FUNCTION_BLOCK POU IMPLEMENTS ITcTask
VAR_INPUT
END_VAR
VAR_OUTPUT
END_VAR
VAR
END_VAR

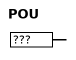
// ???: input not connected

{attribute 'TcTypeSystem'}
{attribute 'no-analysis'}
{attribute 'c++_compatible'}
{attribute 'minimal_input_size' := '4'}
{attribute 'pack_mode' := '4'}
{warning 'add method implementation '}
METHOD GetCurrentDcTime : HRESULT
VAR_INPUT
	pDcTime	: POINTER TO UDINT;
END_VAR
END_METHOD

{attribute 'TcTypeSystem'}
{attribute 'no-analysis'}
{attribute 'c++_compatible'}
{attribute 'minimal_input_size' := '4'}
{attribute 'pack_mode' := '4'}
{warning 'add method implementation '}
METHOD GetCurrentSysTime : HRESULT
VAR_INPUT
	pSysTime	: POINTER TO ULINT;
END_VAR
END_METHOD

{attribute 'TcTypeSystem'}
{attribute 'no-analysis'}
{attribute 'c++_compatible'}
{attribute 'minimal_input_size' := '4'}
{attribute 'pack_mode' := '4'}
{warning 'add method implementation '}
METHOD GetCycleCounter : HRESULT
VAR_INPUT
	pCnt	: POINTER TO ULINT;
END_VAR
END_METHOD

{attribute 'TcTypeSystem'}
{attribute 'no-analysis'}
{attribute 'c++_compatible'}
{attribute 'minimal_input_size' := '4'}
{attribute 'pack_mode' := '4'}
{warning 'add method implementation '}
METHOD GetCycleTime : HRESULT
VAR_INPUT
	pCycleTimeNS	: POINTER TO UDINT;
END_VAR
END_METHOD

{attribute 'TcTypeSystem'}
{attribute 'no-analysis'}
{attribute 'c++_compatible'}
{attribute 'minimal_input_size' := '4'}
{attribute 'pack_mode' := '4'}
{warning 'add method implementation '}
METHOD GetPriority : HRESULT
VAR_INPUT
	pPriority	: POINTER TO UDINT;
END_VAR
END_METHOD

{attribute 'TcTypeSystem'}
{attribute 'no-analysis'}
{attribute 'c++_compatible'}
{attribute 'minimal_input_size' := '4'}
{attribute 'pack_mode' := '4'}
{warning 'add method implementation '}
METHOD TcAddRef : UDINT
END_METHOD

{attribute 'TcTypeSystem'}
{attribute 'no-analysis'}
{attribute 'c++_compatible'}
{attribute 'minimal_input_size' := '4'}
{attribute 'pack_mode' := '4'}
{warning 'add method implementation '}
METHOD TcQueryInterface : HRESULT
VAR_INPUT
	iid	: REFERENCE TO IID;
	pipItf	: POINTER TO PVOID;
END_VAR
END_METHOD

{attribute 'TcTypeSystem'}
{attribute 'no-analysis'}
{attribute 'c++_compatible'}
{attribute 'minimal_input_size' := '4'}
{attribute 'pack_mode' := '4'}
{warning 'add method implementation '}
METHOD TcRelease : UDINT
END_METHOD

END_FUNCTION_BLOCK

(* stored: Version 1.1.0.1, ProductVersion 3.1.4024.4
   POU POU: Id {65d2d1d8-6ae9-4f21-9e48-7c9767404d1b}, SpecialFunc None
   Method GetCurrentDcTime: Id {de8ed7e5-4799-43ee-a95f-177a2cb275c9}
   Method GetCurrentSysTime: Id {b97cb984-1d0e-425a-8cf9-09347fc52933}
   Method GetCycleCounter: Id {ba787561-95ae-47e7-b403-d7105432fa7e}
   Method GetCycleTime: Id {cd459fc4-2458-4684-ac9a-3f070c51d652}
   Method GetPriority: Id {3ceabd74-a870-4f14-89d9-28880da605e6}
   Method TcAddRef: Id {d0b295a4-2f77-4744-8335-2c26dcdabbc9}
   Method TcQueryInterface: Id {9bdd864e-426f-465a-b7a8-6c154e0901e4}
   Method TcRelease: Id {5174f18e-7353-4c15-81e0-388d09ee9cc7} *)
